# EPICS alarm handler configuration: mps_database/bare/alarms/areas/mpln_dog_mp03.alhConfig
GROUP NULL MPLN:DOG:MP03:1
$ALIAS MPS Link Node 74
$GUIDANCE
LTUH MPS
   Group Name: MPLN:DOG:MP03:1
   Summary PV:  MPLN:DOG:MP03:1:STATSUMY
$END
CHANNEL  MPLN:DOG:MP03:1    MPLN:DOG:MP03:1:MPS_EN_RBV		-----
CHANNEL  MPLN:DOG:MP03:1    MPLN:DOG:MP03:1:LC1_MODE_RBV		-----
